{attribute 'linkalways'} 
{attribute 'no_explicit_call' := 'This FB is a CLASS and must be accessed using methods or properties'}
{attribute 'enable_dynamic_creation'}
FUNCTION_BLOCK Node_F_VN_MedianElementElementwise_TcVnPoint2_DINT EXTENDS VisionNode
VAR
    ipContainer : _ITcVnContainer;
    aMedian : _TcVnPoint2_DINT;
    hrPrev : _HRESULT(S_OK);
    hresult : _HRESULT(S_OK);
END_VAR

METHOD PUBLIC  Clone : I_Node
VAR
	pNode : POINTER TO Node_F_VN_MedianElementElementwise_TcVnPoint2_DINT;
END_VAR
pNode := __NEW(Node_F_VN_MedianElementElementwise_TcVnPoint2_DINT);
Clone := pNode^;
END_METHOD

METHOD FB_init : BOOL
VAR_INPUT
	bInitRetains : BOOL; // if TRUE, the retain variables are initialized (warm start / cold start)
	bInCopyCode : BOOL;  // if TRUE, the instance afterwards gets moved into the copy code (online change)
END_VAR
AddInput('ipContainer', ipContainer);
AddInput('aMedian', aMedian);
AddInput('hrPrev', hrPrev);
AddOutput('ipContainer', ipContainer);
AddOutput('hresult',hresult);
END_METHOD

METHOD PROTECTED OnExecute : HRESULT
hresult.Value := F_VN_MedianElementElementwise_TcVnPoint2_DINT(
    ipContainer := ipContainer.Value,
    aMedian := aMedian.Value,
    hrPrev:= hrPrev.Value);
END_METHOD

METHOD PUBLIC PreExecutionCheck
VAR_INPUT
	Check : I_PreExecutionChecks;
END_VAR
Check.IsTrue(ipContainer.IsValid, 'ipContainer must be a valid container');
END_METHOD

END_FUNCTION_BLOCK

(* stored: Version 1.1.0.1, ProductVersion 3.1.4024.13
   POU Node_F_VN_MedianElementElementwise_TcVnPoint2_DINT: Id {1dd2ad6c-e20d-4301-9a2e-9bbc6af88e09}, SpecialFunc None
   Folder Constructor: Id {2e7ca649-a8ff-4073-8b69-fb5296d3674d}
   Method Clone: Id {ad1e40a5-52e8-4c1e-8d90-6b0b19c18530}
   Method FB_init: Id {5b1d500d-68bc-45ba-ae2a-dcf2c7ec9fb1}
   Method OnExecute: Id {db819edc-9814-4b70-af58-87fba372c4a4}
   Method PreExecutionCheck: Id {99e9c415-490f-4406-a918-e8b1df23706b} *)
